{attribute 'linkalways'} 
{attribute 'no_explicit_call' := 'This FB is a CLASS and must be accessed using methods or properties'}
{attribute 'enable_dynamic_creation'}
FUNCTION_BLOCK Node_F_VN_ContourArea EXTENDS VisionNode
VAR
    ipContour : _ITcVnContainer;
    fArea : _LREAL(0.0);
    hrPrev : _HRESULT(S_OK);
	hresult : _HRESULT(S_OK);
END_VAR

METHOD PUBLIC  Clone : I_Node
VAR
	pNode : POINTER TO Node_F_VN_ContourArea;
END_VAR
pNode := __NEW(Node_F_VN_ContourArea);
Clone := pNode^;
END_METHOD

METHOD FB_init : BOOL
VAR_INPUT
	bInitRetains : BOOL; // if TRUE, the retain variables are initialized (warm start / cold start)
	bInCopyCode : BOOL;  // if TRUE, the instance afterwards gets moved into the copy code (online change)
END_VAR
AddInput('ipContour', ipContour);
AddInput('hrPrev', hrPrev);
AddOutput('fArea', fArea);
AddOutput('hresult',hresult);
END_METHOD

METHOD PROTECTED OnExecute
hresult.Value := F_VN_ContourArea(
	ipContour := ipContour.Value,
    fArea := fArea.Value,
	hrPrev:= hrPrev.Value);
END_METHOD

METHOD PUBLIC PreExecutionCheck
VAR_INPUT
	Check : I_PreExecutionChecks;
END_VAR
Check.IsTrue(ipContour.IsValid, 'ipContour must be a valid container');
Check.IsTrue((ipContour.IsType(TC_GLOBAL_CONST_LIST.ContainerType_Vector_TcVnPoint2_DINT) OR
              ipContour.IsType(TC_GLOBAL_CONST_LIST.ContainerType_Vector_TcVnPoint2_REAL)),
              'ipContour contains incorrect type');
END_METHOD

END_FUNCTION_BLOCK

(* stored: Version 1.1.0.1, ProductVersion 3.1.4026.13
   POU Node_F_VN_ContourArea: Id {b09f4f30-7cf7-0d06-3c35-56475c319e24}, SpecialFunc None
   Folder Constructor: Id {0b8e346a-814a-027a-3c78-03e1fe53a346}
   Method Clone: Id {72cf0661-eb93-0960-3463-0c4fef8f07e3}
   Method FB_init: Id {9fd1e84c-c259-0eb5-3b15-a30dd145c7c5}
   Method OnExecute: Id {80976bac-6baa-033e-03b6-5475f859b4d9}
   Method PreExecutionCheck: Id {d0c7115a-7360-00aa-15d8-dade9d093f17} *)
